TYPE UnitTestStructGroup :
STRUCT
	TestBool	: BOOL;
	TestInt		: INT;
	TestReal	: REAL;
END_STRUCT
END_TYPE

(* stored: Version 1.1.0.1, ProductVersion 3.1.4024.11
   DUT UnitTestStructGroup: Id {9b1cc4d3-65cf-41a3-a79d-91a7377f9008} *)
